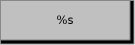
VISUALIZATION ButtonGreenInd  // 135x45
VAR_IN_OUT
	m_Input_ValueTag : None;
END_VAR
VAR_IN_OUT
	m_Input_AssignValue : None;
END_VAR
VAR_IN_OUT
	m_Input_Text : None;
END_VAR
VAR_IN_OUT
	m_Input_ColourTag : None;
END_VAR
VAR_IN_OUT
	m_Input_TapTag : None;
END_VAR
    Rectangle (1,1 132x42)
    Rectangle (0,0 130x40), "%s", text variable: m_Input_Text, colour toggle: (m_Input_ColourTag) <> 0
        tap m_Input_TapTag
        OnMouseUp: execute { m_Input_ValueTag:=(m_Input_AssignValue); }
END_VISUALIZATION

(* stored: Version 1.1.0.1, ProductVersion 3.1.4018.2
   Visu ButtonGreenInd: Id {e8c72a8b-ab6a-45a6-9555-054bd4856ce9} *)
